INTERFACE I_DigitalInput EXTENDS I_Component, I_ForcibleBool

{attribute 'monitoring' := 'call'}
PROPERTY IsActive : BOOL
GET
END_GET
END_PROPERTY

END_INTERFACE

(* stored: Version 1.1.0.1, ProductVersion 3.1.4026.18
   Itf I_DigitalInput: Id {97751258-1f05-41a4-a520-e408a0b73453}
   Property IsActive: Id {8ac2984a-a273-4be2-9eac-24c8c5948a52}
   Get Get: Id {e3fa412e-f7bb-4280-94ff-7281ec25f823} *)
